(* CODESYS project Project_2_RECOVERED_2024-11-26T06-58-48.project

Project tree, tasks and I/O mapping:
  Device : CODESYS Control Win V3 x64, CODESYS, version 3.5.20.30
    application Application
      libraries: Standard, 3.5.18.0 (System); CmpBitmapPool, * (System); Util, 3.5.19.0 (System); VisuDialogs, * (System)
      task MainTask (cyclic, interval t#20ms, priority 1) calls MainPage
      task VISU_TASK (cyclic, interval 100 ms, priority 31) calls VisuElems.Visu_Prg
      function block Timer [LD]
      function block FSM [ST]
      image pool iImages
      function block DosingBlock [ST]
      program MainPage [CFC]: Animation
      program PLC_PRG [CFC]
      visualisation Visualization
      function block Lamps [ST]
  text list GlobalTextList
*)

// Device/Application/MainPage
PROGRAM MainPage
VAR
	// Digital Output
	Elev1_coil    : BOOL;
	Elev2_coil    : BOOL;
	Spiral1_coil  : BOOL;
	Spiral2_coil  : BOOL;
	MixerCoil     : BOOL;
    Gate          : BOOL;
	Blue_Light		: BOOL;
	

	// Digital Input
	Elev1_OVLD    : BOOL;
	ELev2_OVLD    : BOOL;
	Spiral_VFD_OVLD  : BOOL;
	Spira2_VFD_OVLD  : BOOL;
    Mixer_VFD_OVLD   : BOOL;
	Emergency		: BOOL;
	RESET		: BOOL;
	
	
	// Analog Output
	Spiral1_freq  : INT;
	Spiral2_freq  : INT;
	Mixer_freq    : INT;
	
	
	// Analog Input
	Silo1_weight   : INT;
	Silo2_weight   : INT;
	
	// Others
	Start_Dosing      : BOOL;
	Stop_Dosing       : BOOL;
	Fill_Silo1        : BOOL;
	Fill_Silo2        : BOOL;
	
	Silo1_Required    : INT;
	Silo2_Required    : INT;
	
	Dosing_Block: DosingBlock;
	DosingBlockSilo1: DosingBlock;
	DosingBlock1: DosingBlock;
	DosingBlock2: DosingBlock;
	MainController: FSM;
	TimerActivation: Timer;
	Silo_1: LIN_TRAFO;
	Silo1Animation: WORD;
	Silo1AnimationScale: WORD;
	Silo_2: LIN_TRAFO;
	Silo2Animation: WORD;
	Silo2AnimationScale: WORD;
	OVERLOAD: BOOL;
	TON_0: TON;
	Blinker: TON;
	Blinker_Counter: CTU;
	MixerBladeAnimation: WORD;
	GateTimerDone: BOOL;
	LampsBlock: Lamps;
	OVLDorEMGC: BOOL;
	Working: BOOL;
	Done: BOOL;
	LampsBock: Lamps;
	NotEnough: BOOL;
END_VAR
VAR // added by the converter: edge detectors and wires of the graphical bodies
    _w1 : BOOL;
END_VAR

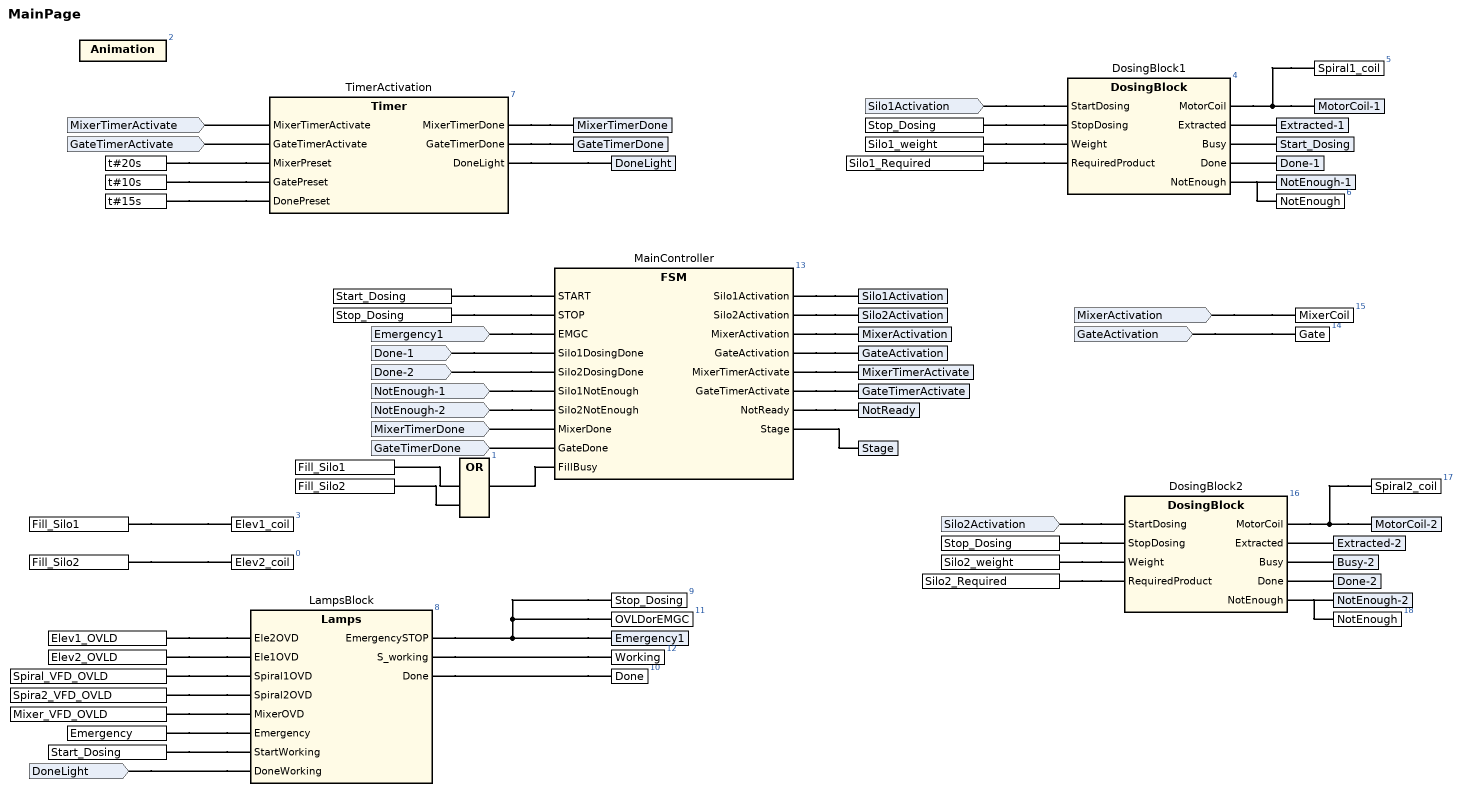
Elev2_coil := Fill_Silo2;
_w1 := Fill_Silo1 OR Fill_Silo2;
Animation();
Elev1_coil := Fill_Silo1;
DosingBlock1(
    StartDosing := MainController.Silo1Activation,
    StopDosing := Stop_Dosing,
    Weight := Silo1_weight,
    RequiredProduct := Silo1_Required); // DosingBlock
Spiral1_coil := DosingBlock1.MotorCoil;
NotEnough := DosingBlock1.NotEnough;
TimerActivation(
    MixerTimerActivate := MainController.MixerTimerActivate,
    GateTimerActivate := MainController.GateTimerActivate,
    MixerPreset := t#20s,
    GatePreset := t#10s,
    DonePreset := t#15s); // Timer
LampsBlock(
    Ele2OVD := Elev1_OVLD,
    Ele1OVD := Elev2_OVLD,
    Spiral1OVD := Spiral_VFD_OVLD,
    Spiral2OVD := Spira2_VFD_OVLD,
    MixerOVD := Mixer_VFD_OVLD,
    Emergency := Emergency,
    StartWorking := Start_Dosing,
    DoneWorking := TimerActivation.DoneLight); // Lamps
Stop_Dosing := LampsBlock.EmergencySTOP;
Done := LampsBlock.Done;
OVLDorEMGC := LampsBlock.EmergencySTOP;
Working := LampsBlock.S_working;
MainController(
    START := Start_Dosing,
    STOP := Stop_Dosing,
    EMGC := LampsBlock.EmergencySTOP,
    Silo1DosingDone := DosingBlock1.Done,
    Silo2DosingDone := DosingBlock2.Done,
    Silo1NotEnough := DosingBlock1.NotEnough,
    Silo2NotEnough := DosingBlock2.NotEnough,
    MixerDone := TimerActivation.MixerTimerDone,
    GateDone := TimerActivation.GateTimerDone,
    FillBusy := _w1); // FSM
Gate := MainController.GateActivation;
MixerCoil := MainController.MixerActivation;
DosingBlock2(
    StartDosing := MainController.Silo2Activation,
    StopDosing := Stop_Dosing,
    Weight := Silo2_weight,
    RequiredProduct := Silo2_Required); // DosingBlock
Spiral2_coil := DosingBlock2.MotorCoil;
NotEnough := DosingBlock2.NotEnough;

ACTION Animation:
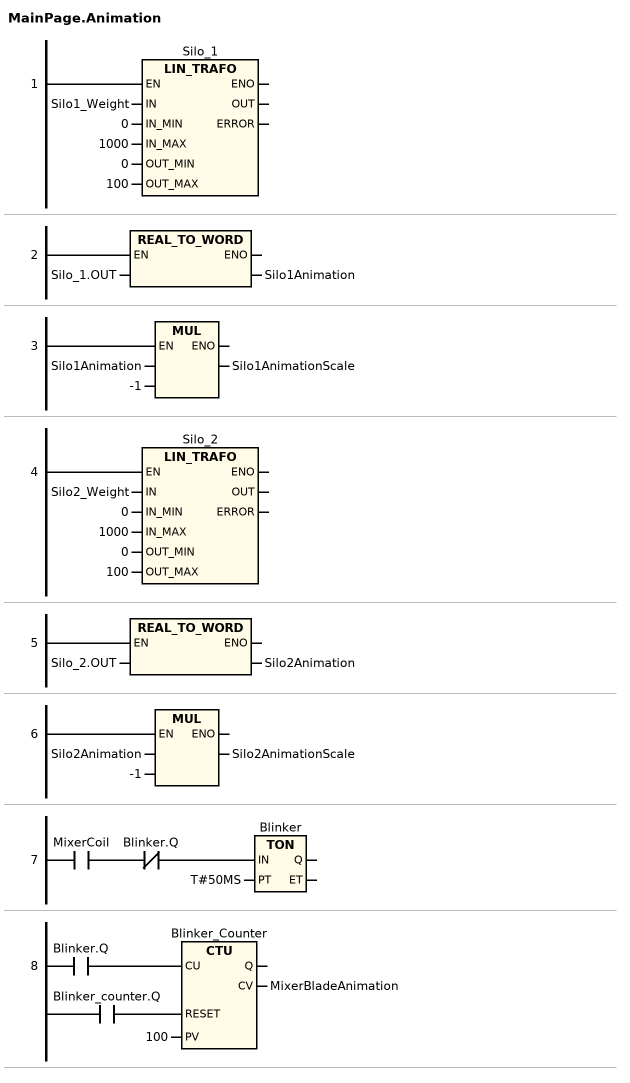
// NETWORK 1
Silo_1(IN := Silo1_Weight, IN_MIN := 0, IN_MAX := 1000, OUT_MIN := 0, OUT_MAX := 100); // LIN_TRAFO

// NETWORK 2
Silo1Animation := REAL_TO_WORD(Silo_1.OUT);

// NETWORK 3
Silo1AnimationScale := Silo1Animation * -1;

// NETWORK 4
Silo_2(IN := Silo2_Weight, IN_MIN := 0, IN_MAX := 1000, OUT_MIN := 0, OUT_MAX := 100); // LIN_TRAFO

// NETWORK 5
Silo2Animation := REAL_TO_WORD(Silo_2.OUT);

// NETWORK 6
Silo2AnimationScale := Silo2Animation * -1;

// NETWORK 7
Blinker(IN := MixerCoil AND NOT Blinker.Q, PT := T#50MS); // TON

// NETWORK 8
Blinker_Counter(CU := Blinker.Q, RESET := Blinker_counter.Q, PV := 100, CV => MixerBladeAnimation); // CTU
END_ACTION

END_PROGRAM

// Device/Application/DosingBlock
FUNCTION_BLOCK DosingBlock

VAR_INPUT
	StartDosing   : BOOL;
	StopDosing    : BOOL;
	Weight        : INT;
	RequiredProduct : INT;
	
END_VAR

VAR_OUTPUT
	MotorCoil    : BOOL;
	Extracted    : INT;
	Busy         : BOOL;
	Done         : BOOL;
	NotEnough    : BOOL;
	
END_VAR

VAR
	Weight_saved  : INT;
	StartTrig : R_TRIG;
	

END_VAR

StartTrig(CLK:=StartDosing , Q=> );

IF StartTrig.Q = 1 AND NotEnough = 0  AND StopDosing = 0 THEN
	Weight_saved := Weight;
	MotorCoil := 1;
	Busy := 1;
	Done := 0;	
END_IF

IF Busy =1 THEN
	Extracted := Weight_saved - Weight;
	IF Extracted >= RequiredProduct THEN
		MotorCoil := 0;
		Busy      := 0;
		Done	  := 1; 
	END_IF
END_IF


IF RequiredProduct > Weight AND Busy = 0 THEN
	NotEnough   := 1;
ELSE
	NotEnough	:= 0;
END_IF


IF StopDosing = 1 THEN
	MotorCoil := 0;
	Busy      := 0;
	Done	  := 1;	
END_IF

END_FUNCTION_BLOCK

// Device/Application/Timer
FUNCTION_BLOCK Timer
VAR_INPUT
	MixerTimerActivate	:BOOL;
	GateTimerActivate	:BOOL;
	MixerPreset			: TIME;
	GatePreset			: TIME;
	DonePreset: TIME;
	
END_VAR

VAR_OUTPUT
	MixerTimerDone		:BOOL;
	GateTimerDone		:BOOL;
	DoneLight: BOOL;
END_VAR
VAR
	GateTimer: TON;
	MixerTimer: TON;

	
	Done: TOF;
	
END_VAR

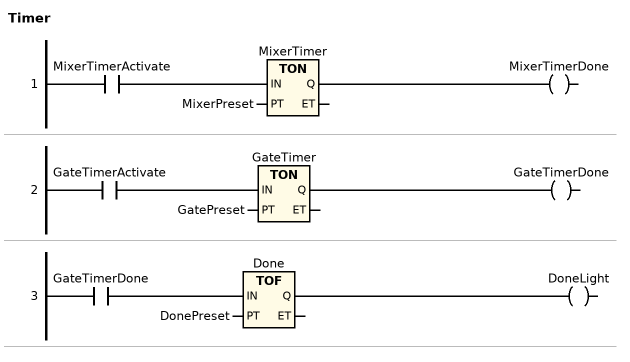
// NETWORK 1
MixerTimer(IN := MixerTimerActivate, PT := MixerPreset); // TON
MixerTimerDone := MixerTimer.Q;

// NETWORK 2
GateTimer(IN := GateTimerActivate, PT := GatePreset); // TON
GateTimerDone := GateTimer.Q;

// NETWORK 3
Done(IN := GateTimerDone, PT := DonePreset); // TOF
DoneLight := Done.Q;

END_FUNCTION_BLOCK

// Device/Application/Lamps
FUNCTION_BLOCK Lamps
VAR_INPUT
	Spiral1OVD		: BOOL;
	Spiral2OVD		: BOOL;
	MixerOVD		: BOOL;
	Ele1OVD			: BOOL;
	Ele2OVD			: BOOL;
	Emergency		: BOOL;
	StartWorking     : BOOL;
	DoneWorking		: BOOL;
	
END_VAR



VAR_OUTPUT
	EmergencySTOP		:BOOL;
	S_working		:BOOL;
	Done		:BOOL;
	
END_VAR
VAR
	StartWorkingTrig: R_TRIG;
END_VAR

StartWorkingTrig(CLK:=StartWorking , Q=> );
IF StartWorkingTrig.Q=1 THEN
	S_working :=1;
END_IF

IF DoneWorking =1 THEN
	Done := 1;
	S_working := 0;
ELSE
	Done:=0;
END_IF

IF Spiral1OVD =1 OR Spiral2OVD = 1 OR MixerOVD = 1  OR Ele1OVD = 1 OR Ele2OVD =1 OR  Emergency =1 THEN
	EmergencySTOP:= 1;
	S_working := 0;
	Done:=0;
ELSE
	EmergencySTOP:=0;

END_IF

END_FUNCTION_BLOCK

// Device/Application/FSM
FUNCTION_BLOCK FSM

VAR_INPUT
	START	: BOOL;
	STOP	: BOOL;
	EMGC	: BOOL;
	Silo1DosingDone	: BOOL;
	Silo2DosingDone	: BOOL;
	Silo1NotEnough	: BOOL;
	Silo2NotEnough	: BOOL;
	MixerDone		: BOOL;
	GateDone		: BOOL;
	FillBusy	: BOOL;
END_VAR

VAR_OUTPUT
	Silo1Activation		: BOOL;
	Silo2Activation 	: BOOL;
	MixerActivation		: BOOL;
	GateActivation		: BOOL;
	MixerTimerActivate	: BOOL;
	GateTimerActivate	: BOOL;
	NotReady			: BOOL;
	Stage				: INT;
END_VAR

VAR
	StartTrigger : R_TRIG;
	Silo1_TRIG : R_TRIG;
	Silo2_TRIG : R_TRIG;
END_VAR

StartTrigger(CLK:=START , Q=> );
Silo1_TRIG(CLK:=Silo1DosingDone , Q=> );
Silo2_TRIG(CLK:=Silo2DosingDone , Q=> );
CASE Stage OF
0:
IF StartTrigger.Q = 1 AND NotReady=0 THEN 
	Stage := 1;
END_IF

IF Silo1NotEnough OR Silo2NotEnough THEN
	NotReady := 1;
    Silo1Activation := 0;
    Silo2Activation := 0;
    MixerActivation := 0;
    GateActivation := 0;
    MixerTimerActivate := 0;
    GateTimerActivate := 0;
    Stage := 0; // Remain in Stage 0
END_IF 
	
1:
Silo1Activation := 1;

IF Silo1_TRIG.Q = 1 THEN
	Silo1Activation:= 0;
	Stage:= 2;
END_IF

	
2:
Silo2Activation:= 1;
	
IF Silo2_TRIG.Q = 1 THEN
	Silo2Activation:= 0;
	Stage:= 3;
END_IF	

	
	
3:
MixerActivation:= 1;
MixerTimerActivate:=1;
IF 	MixerDone = 1 THEN 
	MixerActivation:= 0;
	MixerTimerActivate:=0;
	Stage:= 4;
END_IF
	
	
4:
GateActivation:= 1;
GateTimerActivate:=1;
IF 	GateDone = 1 THEN 
	GateActivation:= 0;
	GateTimerActivate:=0;
	Stage:= 0;	
END_IF		
END_CASE


IF EMGC  OR  STOP   OR FillBusy THEN
	NotReady 	:= 1;
	Silo1Activation	:= 0;
	Silo2Activation	:= 0;
	MixerActivation	:= 0;
	GateActivation	:=  0;
	MixerTimerActivate	:=0;
	GateTimerActivate	:=0;
	Stage:=0;
	
ELSE
	NotReady:= 0;
END_IF

END_FUNCTION_BLOCK

// Device/Application/PLC_PRG
PROGRAM PLC_PRG
VAR
END_VAR

END_PROGRAM

// Device/Application/Visualization
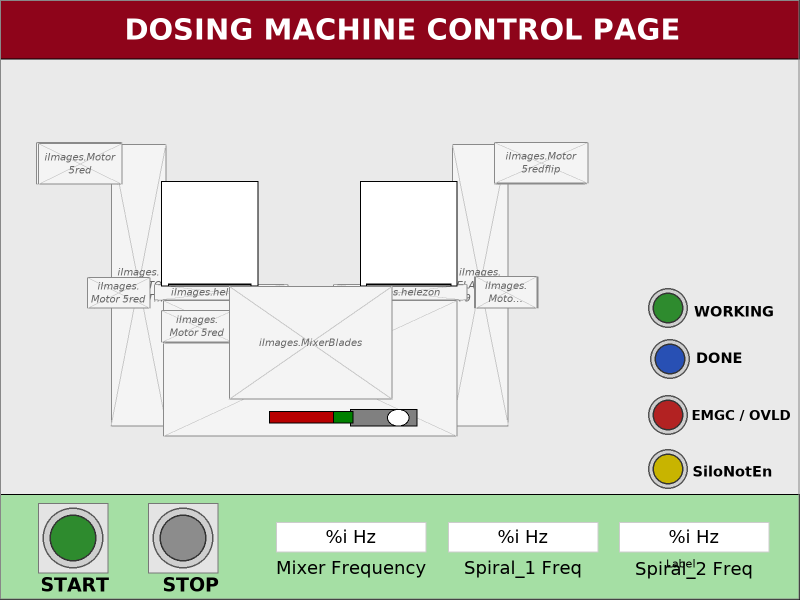
VISUALIZATION Visualization  // 800x600
    Rectangle (0,0 800x59)
    Rectangle (0,494 800x106)
    Label (5,0 795x59), "DOSING MACHINE CONTROL PAGE"
    PushSwitch (38,503 70x70), variable: MainPage.Start_Dosing, behaviour: TAP, style: Switch-PushSwitch-Green
    PushSwitch (148,503 70x70), variable: MainPage.Stop_Dosing, behaviour: TAP, style: Switch-PushSwitch-Gray
    Textfield (276,522 150x30), "%i Hz", text variable: MainPage.Mixer_freq
        OnMouseClick: write the text variable via Default, min 0, max 60
    Textfield (448,522 150x30), "%i Hz", text variable: MainPage.Spiral1_freq
        OnMouseClick: write the text variable via Default, min 0, max 60
    Textfield (619,522 150x30), "%i Hz", text variable: MainPage.Spiral2_freq
        OnMouseClick: write the text variable via Default, min 0, max 60
    Label (276,553 150x30), "Mixer Frequency"
    Label (448,553 150x30), "Spiral_1 Freq"
    Label (681,562 0x4), "Label"
    Label (619,554 150x30), "Spiral_2 Freq"
    Label (0,570 150x30), "START"
    Label (116,570 150x30), "STOP"
    Image (111,144 55x282), image: iImages.ELAVATOR 9 METRE - Kopya
    Image (452,144 56x282), image: iImages.ELAVATOR 9 METREFlip
    Image (333,284 134x16), image: iImages.helezon
    Image (154,284 134x16), image: iImages.helezonFlip
    Rectangle (161,181 97x105)
    Rectangle (360,181 97x105)
    Image (163,300 294x136), image: iImages.Silo
    RoundedRectangle (168,284 83x0)
        p2773130477: MainPage.Silo1AnimationScale
    RoundedRectangle (366,284 85x0)
        p2773130477: MainPage.Silo2AnimationScale
    Image (36,144 81x40), image: iImages.Motor 5
    Image (36,142 86x42), invisible if: MainPage.Elev1_coil = 0, image: iImages.Motor 5green
    Image (38,143 84x41), invisible if: MainPage.Elev1_OVLD=0, image: iImages.Motor 5red
    Image (163,310 68x33), image: iImages.Motor 5
    Image (161,310 67x32), invisible if: MainPage.MixerCoil=0, image: iImages.Motor 5green
    Image (161,310 72x32), invisible if: MainPage.Mixer_VFD_OVLD=0, image: iImages.Motor 5red
    Image (498,142 88x42), image: iImages.Motor 5Flip
    Image (494,144 92x40), invisible if: MainPage.Elev2_coil = 0, image: iImages.Motor 5greenFlip
    Image (494,142 94x41), invisible if: MainPage.ELev2_OVLD=0, image: iImages.Motor 5redflip
    Lamp1 (645,391 46x48), variable: MainPage.OVLDorEMGC, style: Lamp-Lamp1-Red
    Lamp1 (645,284 46x48), variable: MainPage.Working, style: Lamp-Lamp1-Green
    Image (94,277 56x31), image: iImages.Motor 5
    Image (87,277 63x31), invisible if: MainPage.Spiral1_coil=0, image: iImages.Motor 5green
    Image (87,277 63x31), invisible if: MainPage.Spiral_VFD_OVLD=0, image: iImages.Motor 5red
    Label (698,409 86x13), "EMGC / OVLD"
    Label (701,449 80x13)
    Label (698,299 80x15)
    Image (229,286 163x113), image: iImages.MixerBlades
        p2858320360: MainPage.MixerBladeAnimation
    Rectangle (269,411 84x12), invisible if: MainPage.Gate
    RoundedRectangle (350,409 67x17)
    Ellipse (387,409 22x17)
    Image (477,279 61x29), image: iImages.Motor 5Flip
    Image (474,276 64x32), invisible if: MainPage.Spiral2_coil=0, image: iImages.Motor 5greenFlip
    Image (475,276 62x32), invisible if: MainPage.Spira2_VFD_OVLD=0, image: iImages.Motor 5redflip
    Rectangle (333,411 20x12), invisible if: MainPage.Gate=0
    Lamp1 (647,335 46x48), variable: MainPage.Done, style: Lamp-Lamp1-Blue
    Label (692,343 55x30), "DONE"
    Label (699,299 70x25), "WORKING"
    Lamp1 (645,445 46x48), variable: MainPage.NotEnough, style: Lamp-Lamp1-Yellow
    Label (681,459 103x25), "SiloNotEn"
END_VISUALIZATION
